Staubli VAL3: FlagStatus.dtx

public num ForceFlag
public num RosFlag
public num RobotFlag
